(* Logix 5000 project; controller Lab8_1 5069-L306ERM rev 35.11; software revision 35.03 *)

TASK MainTask (continuous, watchdog 500 ms) : MainProgram

MODULES
   Local : 5069-L306ERM (5069 0, rev 35.11)
      IOHub : vendor 1 type 7 code 358 (Ethernet 192.168.105.5, rev 1.1, Output RPI 20 ms)
END_MODULES

PROGRAM MainProgram   (* main routine Lab8_1 *)
VAR
   i : DINT;
   MrArray : DINT[3];
   MrString : STRING;
END_VAR

ROUTINE Lab8_1   (* structured text *)
   if IOHub:I.Data.0 then
   	for i:= 0 to MrString.LEN by 1 do
   		MrArray[i]:= MrString.DATA[i];
   	end_for;
   	IOHub:O.Data.0:=1;
   end_if;
   
   if IOHub:I.Data.2 then
   	for i:= 0 to MrString.LEN by 1 do
   		MrArray[i]:= 0;
   	end_for;
   	IOHub:O.Data.0:= 0;
   end_if;
END_ROUTINE
END_PROGRAM
